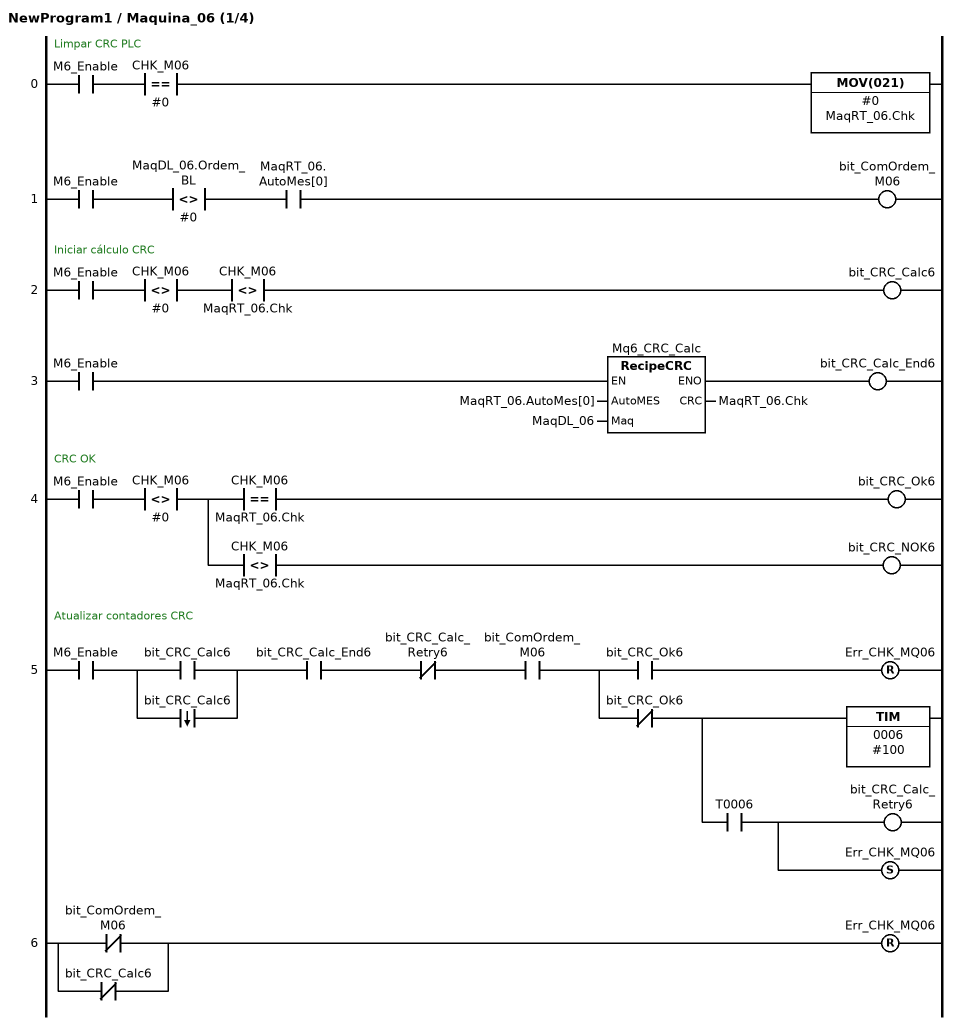
; [picture p24: NewProgram1 / Maquina_06, rungs 0-6]
; rung 0: Limpar CRC PLC
LD M6_Enable
AND=(300) CHK_M06 #0
MOV(021) #0 MaqRT_06.Chk
; rung 1
LD M6_Enable
AND<>L(306) MaqDL_06.Ordem_BL #0
AND MaqRT_06.AutoMes[0]
OUT bit_ComOrdem_M06
; rung 2: Iniciar cálculo CRC
LD M6_Enable
AND<>(305) CHK_M06 #0
AND<>(305) CHK_M06 MaqRT_06.Chk
OUT bit_CRC_Calc6
; rung 3
LD M6_Enable
CALL Mq6_CRC_Calc : RecipeCRC (AutoMES := MaqRT_06.AutoMes[0], Maq := MaqDL_06, CRC => MaqRT_06.Chk)
OUT bit_CRC_Calc_End6
; rung 4: CRC OK
LD M6_Enable
AND<>(305) CHK_M06 #0
OUT TR0
AND=(300) CHK_M06 MaqRT_06.Chk
OUT bit_CRC_Ok6
LD TR0
AND<>(305) CHK_M06 MaqRT_06.Chk
OUT bit_CRC_NOK6
; rung 5: Atualizar contadores CRC
LD M6_Enable
LD bit_CRC_Calc6
%OR bit_CRC_Calc6
ANDLD
AND bit_CRC_Calc_End6
ANDNOT bit_CRC_Calc_Retry6
AND bit_ComOrdem_M06
OUT TR0
AND bit_CRC_Ok6
RSET Err_CHK_MQ06
LD TR0
ANDNOT bit_CRC_Ok6
TIM 0006 #100
AND T0006
OUT bit_CRC_Calc_Retry6
SET Err_CHK_MQ06
; rung 6
LDNOT bit_ComOrdem_M06
ORNOT bit_CRC_Calc6
RSET Err_CHK_MQ06

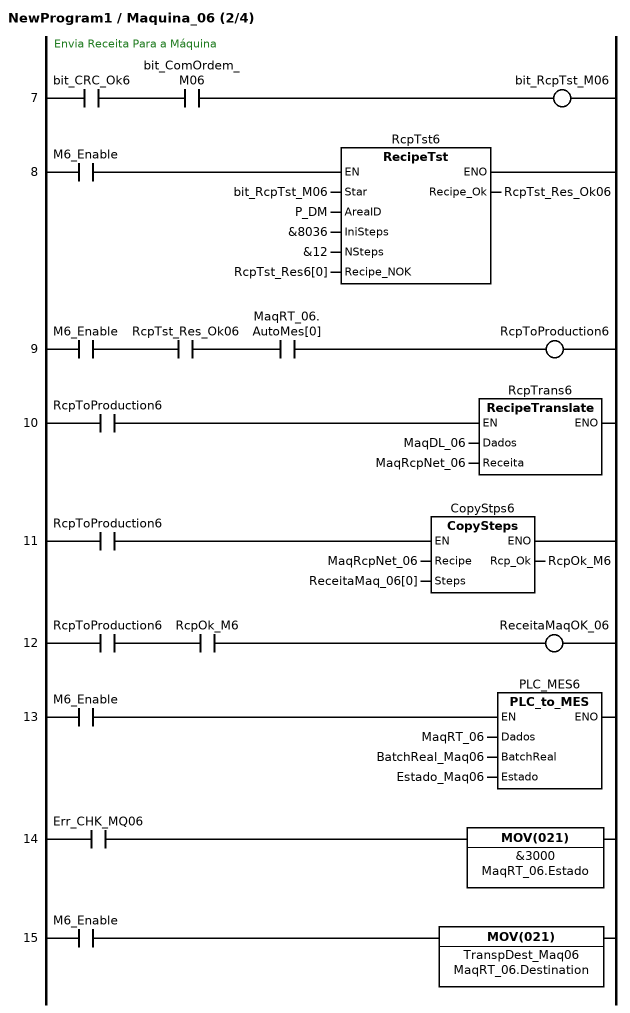
; rung 7: Envia Receita Para a Máquina
LD bit_CRC_Ok6
AND bit_ComOrdem_M06
OUT bit_RcpTst_M06
; rung 8
LD M6_Enable
CALL RcpTst6 : RecipeTst (Star := bit_RcpTst_M06, AreaID := P_DM, IniSteps := &8036, NSteps := &12, Recipe_NOK := RcpTst_Res6[0], Recipe_Ok => RcpTst_Res_Ok06)
; rung 9
LD M6_Enable
AND RcpTst_Res_Ok06
AND MaqRT_06.AutoMes[0]
OUT RcpToProduction6
; rung 10
LD RcpToProduction6
CALL RcpTrans6 : RecipeTranslate (Dados := MaqDL_06, Receita := MaqRcpNet_06)
; rung 11
LD RcpToProduction6
CALL CopyStps6 : CopySteps (Recipe := MaqRcpNet_06, Steps := ReceitaMaq_06[0], Rcp_Ok => RcpOk_M6)
; rung 12
LD RcpToProduction6
AND RcpOk_M6
OUT ReceitaMaqOK_06
; rung 13
LD M6_Enable
CALL PLC_MES6 : PLC_to_MES (Dados := MaqRT_06, BatchReal := BatchReal_Maq06, Estado := Estado_Maq06)
; rung 14
LD Err_CHK_MQ06
MOV(021) &3000 MaqRT_06.Estado
; rung 15
LD M6_Enable
MOV(021) TranspDest_Maq06 MaqRT_06.Destination

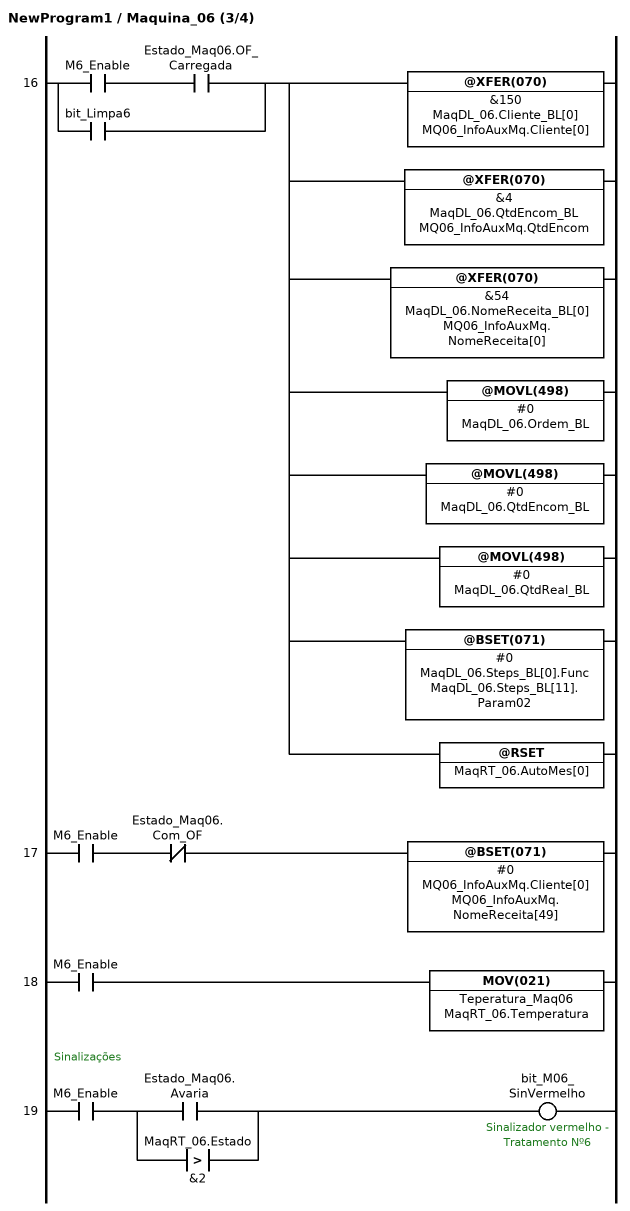
; rung 16
LD M6_Enable
AND Estado_Maq06.OF_Carregada
OR bit_Limpa6
@XFER(070) &150 MaqDL_06.Cliente_BL[0] MQ06_InfoAuxMq.Cliente[0]
@XFER(070) &4 MaqDL_06.QtdEncom_BL MQ06_InfoAuxMq.QtdEncom
@XFER(070) &54 MaqDL_06.NomeReceita_BL[0] MQ06_InfoAuxMq.NomeReceita[0]
@MOVL(498) #0 MaqDL_06.Ordem_BL
@MOVL(498) #0 MaqDL_06.QtdEncom_BL
@MOVL(498) #0 MaqDL_06.QtdReal_BL
@BSET(071) #0 MaqDL_06.Steps_BL[0].Func MaqDL_06.Steps_BL[11].Param02
@RSET MaqRT_06.AutoMes[0]
; rung 17
LD M6_Enable
ANDNOT Estado_Maq06.Com_OF
@BSET(071) #0 MQ06_InfoAuxMq.Cliente[0] MQ06_InfoAuxMq.NomeReceita[49]
; rung 18
LD M6_Enable
MOV(021) Teperatura_Maq06 MaqRT_06.Temperatura
; rung 19: Sinalizações
LD M6_Enable
LD Estado_Maq06.Avaria
OR>(320) MaqRT_06.Estado &2
ANDLD
OUT bit_M06_SinVermelho  ; Sinalizador vermelho - Tratamento Nº6

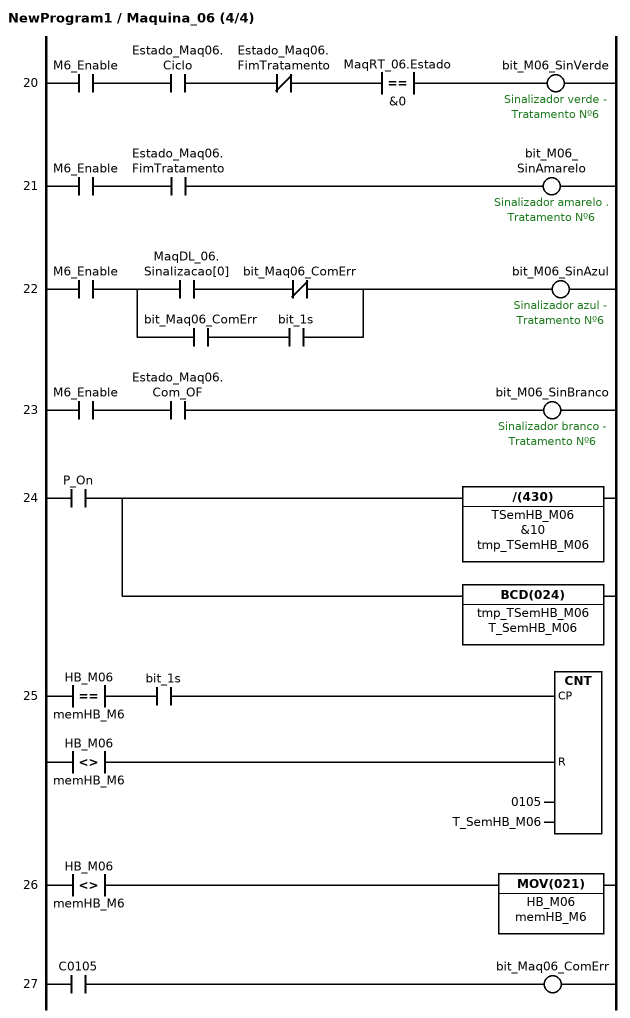
; rung 20
LD M6_Enable
AND Estado_Maq06.Ciclo
ANDNOT Estado_Maq06.FimTratamento
AND=(300) MaqRT_06.Estado &0
OUT bit_M06_SinVerde  ; Sinalizador verde - Tratamento Nº6
; rung 21
LD M6_Enable
AND Estado_Maq06.FimTratamento
OUT bit_M06_SinAmarelo  ; Sinalizador amarelo . Tratamento Nº6
; rung 22
LD M6_Enable
LD MaqDL_06.Sinalizacao[0]
ANDNOT bit_Maq06_ComErr
LD bit_Maq06_ComErr
AND bit_1s
ORLD
ANDLD
OUT bit_M06_SinAzul  ; Sinalizador azul - Tratamento Nº6
; rung 23
LD M6_Enable
AND Estado_Maq06.Com_OF
OUT bit_M06_SinBranco  ; Sinalizador branco - Tratamento Nº6
; rung 24
LD P_On
/(430) TSemHB_M06 &10 tmp_TSemHB_M06
BCD(024) tmp_TSemHB_M06 T_SemHB_M06
; rung 25
LD=(300) HB_M06 memHB_M6
AND bit_1s
LD<>(305) HB_M06 memHB_M6
CNT 0105 T_SemHB_M06
; rung 26
LD<>(305) HB_M06 memHB_M6
MOV(021) HB_M06 memHB_M6
; rung 27
LD C0105
OUT bit_Maq06_ComErr

### Section Maquina_07

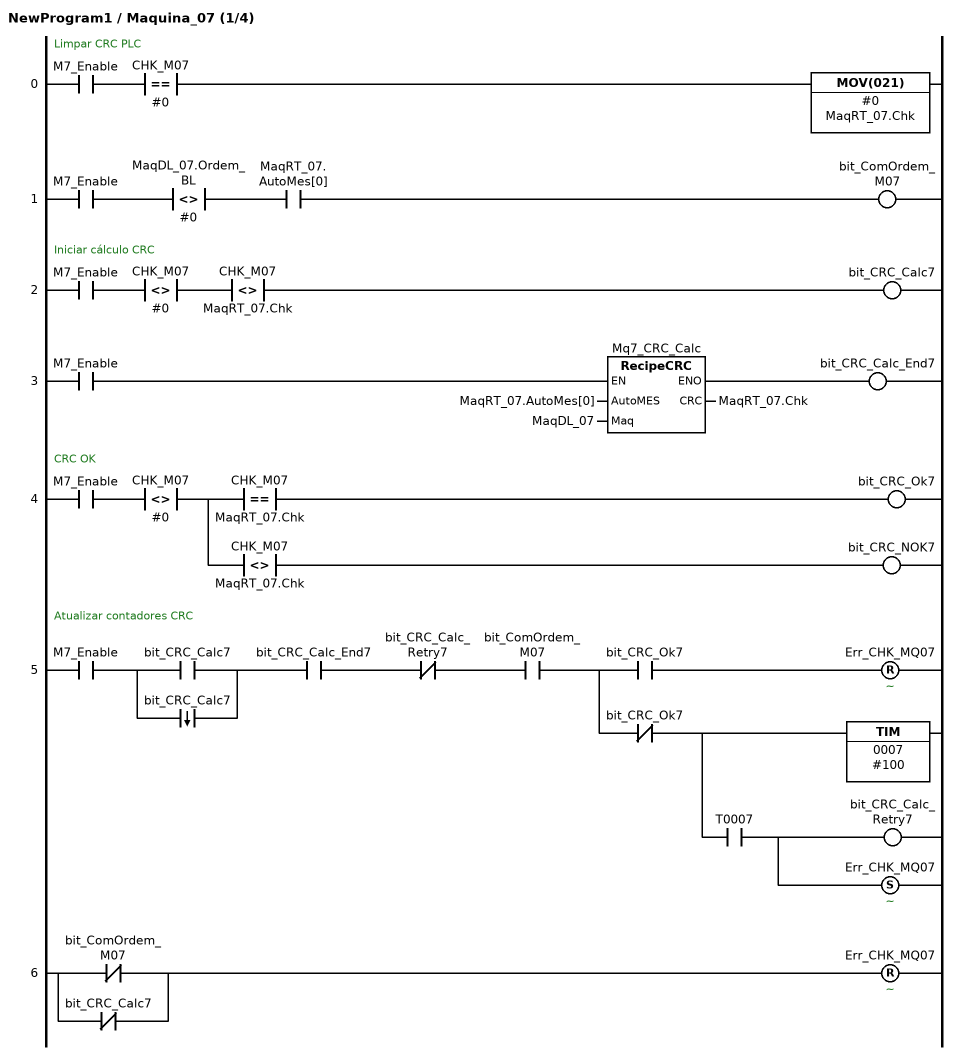
; rung 0: Limpar CRC PLC
LD M7_Enable
AND=(300) CHK_M07 #0
MOV(021) #0 MaqRT_07.Chk
; rung 1
LD M7_Enable
AND<>L(306) MaqDL_07.Ordem_BL #0
AND MaqRT_07.AutoMes[0]
OUT bit_ComOrdem_M07
; rung 2: Iniciar cálculo CRC
LD M7_Enable
AND<>(305) CHK_M07 #0
AND<>(305) CHK_M07 MaqRT_07.Chk
OUT bit_CRC_Calc7
; rung 3
LD M7_Enable
CALL Mq7_CRC_Calc : RecipeCRC (AutoMES := MaqRT_07.AutoMes[0], Maq := MaqDL_07, CRC => MaqRT_07.Chk)
OUT bit_CRC_Calc_End7
; rung 4: CRC OK
LD M7_Enable
AND<>(305) CHK_M07 #0
OUT TR0
AND=(300) CHK_M07 MaqRT_07.Chk
OUT bit_CRC_Ok7
LD TR0
AND<>(305) CHK_M07 MaqRT_07.Chk
OUT bit_CRC_NOK7
; rung 5: Atualizar contadores CRC
LD M7_Enable
LD bit_CRC_Calc7
%OR bit_CRC_Calc7
ANDLD
AND bit_CRC_Calc_End7
ANDNOT bit_CRC_Calc_Retry7
AND bit_ComOrdem_M07
OUT TR0
AND bit_CRC_Ok7
RSET Err_CHK_MQ07  ; ~
LD TR0
ANDNOT bit_CRC_Ok7
TIM 0007 #100
AND T0007
OUT bit_CRC_Calc_Retry7
SET Err_CHK_MQ07  ; ~
; rung 6
LDNOT bit_ComOrdem_M07
ORNOT bit_CRC_Calc7
RSET Err_CHK_MQ07  ; ~

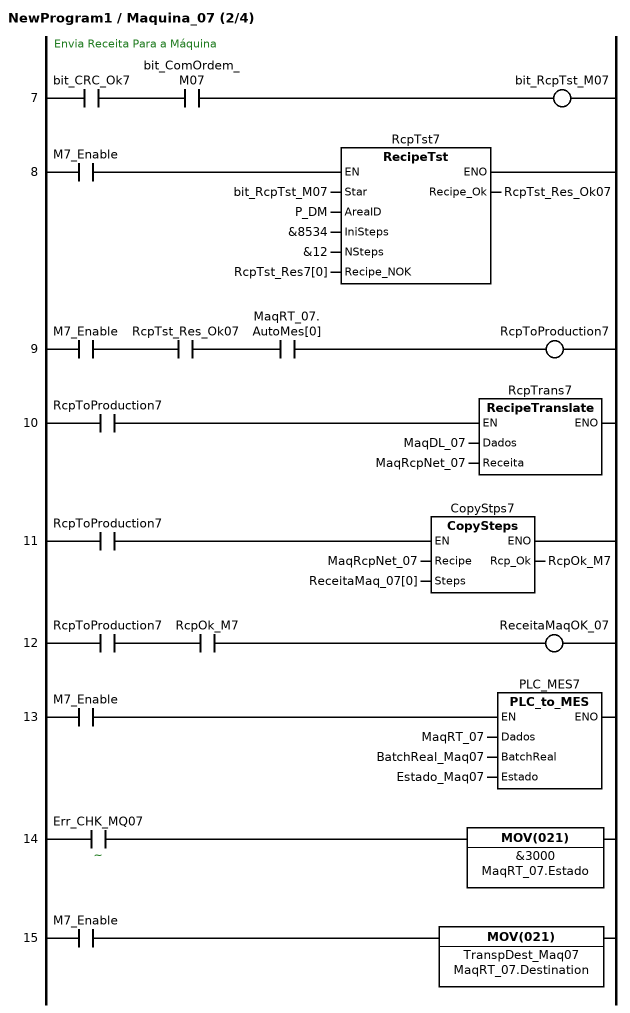
; rung 7: Envia Receita Para a Máquina
LD bit_CRC_Ok7
AND bit_ComOrdem_M07
OUT bit_RcpTst_M07
; rung 8
LD M7_Enable
CALL RcpTst7 : RecipeTst (Star := bit_RcpTst_M07, AreaID := P_DM, IniSteps := &8534, NSteps := &12, Recipe_NOK := RcpTst_Res7[0], Recipe_Ok => RcpTst_Res_Ok07)
; rung 9
LD M7_Enable
AND RcpTst_Res_Ok07
AND MaqRT_07.AutoMes[0]
OUT RcpToProduction7
; rung 10
LD RcpToProduction7
CALL RcpTrans7 : RecipeTranslate (Dados := MaqDL_07, Receita := MaqRcpNet_07)
; rung 11
LD RcpToProduction7
CALL CopyStps7 : CopySteps (Recipe := MaqRcpNet_07, Steps := ReceitaMaq_07[0], Rcp_Ok => RcpOk_M7)
; rung 12
LD RcpToProduction7
AND RcpOk_M7
OUT ReceitaMaqOK_07
; rung 13
LD M7_Enable
CALL PLC_MES7 : PLC_to_MES (Dados := MaqRT_07, BatchReal := BatchReal_Maq07, Estado := Estado_Maq07)
; rung 14
LD Err_CHK_MQ07  ; ~
MOV(021) &3000 MaqRT_07.Estado
; rung 15
LD M7_Enable
MOV(021) TranspDest_Maq07 MaqRT_07.Destination

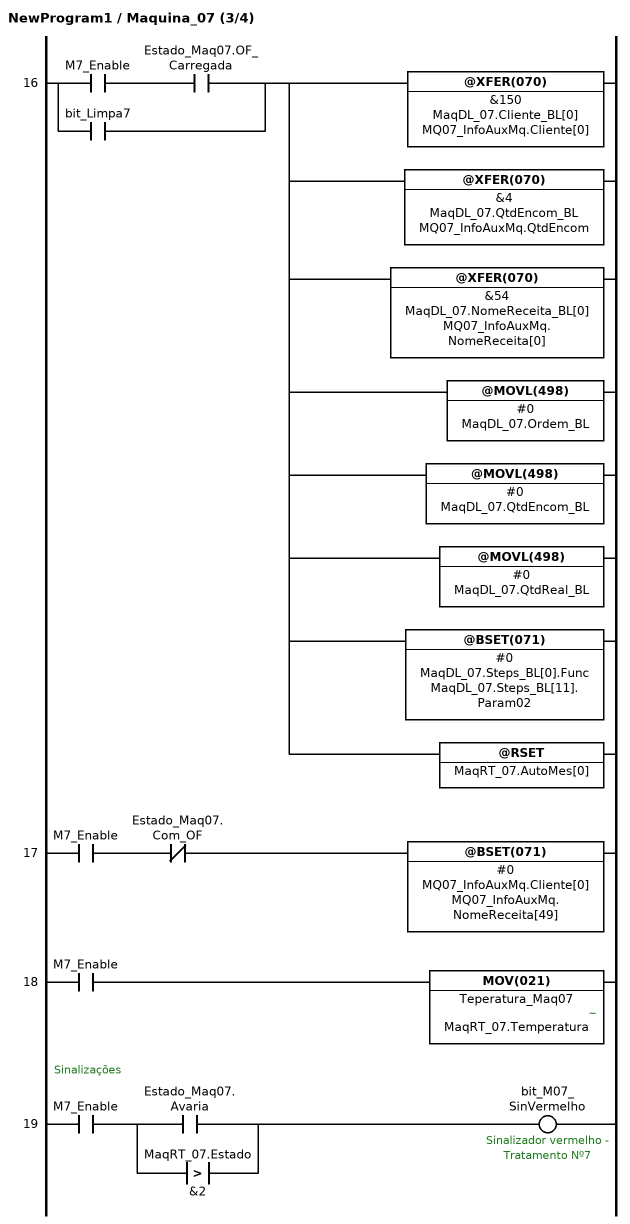
; rung 16
LD M7_Enable
AND Estado_Maq07.OF_Carregada
OR bit_Limpa7
@XFER(070) &150 MaqDL_07.Cliente_BL[0] MQ07_InfoAuxMq.Cliente[0]
@XFER(070) &4 MaqDL_07.QtdEncom_BL MQ07_InfoAuxMq.QtdEncom
@XFER(070) &54 MaqDL_07.NomeReceita_BL[0] MQ07_InfoAuxMq.NomeReceita[0]
@MOVL(498) #0 MaqDL_07.Ordem_BL
@MOVL(498) #0 MaqDL_07.QtdEncom_BL
@MOVL(498) #0 MaqDL_07.QtdReal_BL
@BSET(071) #0 MaqDL_07.Steps_BL[0].Func MaqDL_07.Steps_BL[11].Param02
@RSET MaqRT_07.AutoMes[0]
; rung 17
LD M7_Enable
ANDNOT Estado_Maq07.Com_OF
@BSET(071) #0 MQ07_InfoAuxMq.Cliente[0] MQ07_InfoAuxMq.NomeReceita[49]
; rung 18
LD M7_Enable
MOV(021) Teperatura_Maq07 MaqRT_07.Temperatura  ; ~
; rung 19: Sinalizações
LD M7_Enable
LD Estado_Maq07.Avaria
OR>(320) MaqRT_07.Estado &2
ANDLD
OUT bit_M07_SinVermelho  ; Sinalizador vermelho - Tratamento Nº7

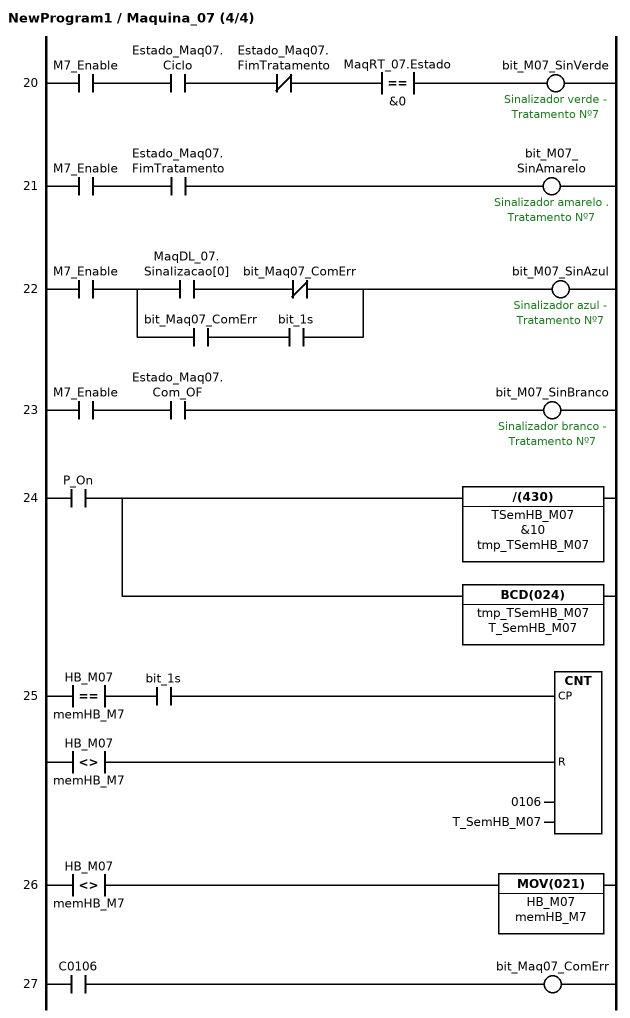
; rung 20
LD M7_Enable
AND Estado_Maq07.Ciclo
ANDNOT Estado_Maq07.FimTratamento
AND=(300) MaqRT_07.Estado &0
OUT bit_M07_SinVerde  ; Sinalizador verde - Tratamento Nº7
; rung 21
LD M7_Enable
AND Estado_Maq07.FimTratamento
OUT bit_M07_SinAmarelo  ; Sinalizador amarelo . Tratamento Nº7
; rung 22
LD M7_Enable
LD MaqDL_07.Sinalizacao[0]
ANDNOT bit_Maq07_ComErr
LD bit_Maq07_ComErr
AND bit_1s
ORLD
ANDLD
OUT bit_M07_SinAzul  ; Sinalizador azul - Tratamento Nº7
; rung 23
LD M7_Enable
AND Estado_Maq07.Com_OF
OUT bit_M07_SinBranco  ; Sinalizador branco - Tratamento Nº7
; rung 24
LD P_On
/(430) TSemHB_M07 &10 tmp_TSemHB_M07
BCD(024) tmp_TSemHB_M07 T_SemHB_M07
; rung 25
LD=(300) HB_M07 memHB_M7
AND bit_1s
LD<>(305) HB_M07 memHB_M7
CNT 0106 T_SemHB_M07
; rung 26
LD<>(305) HB_M07 memHB_M7
MOV(021) HB_M07 memHB_M7
; rung 27
LD C0106
OUT bit_Maq07_ComErr

### Section Maquina_08

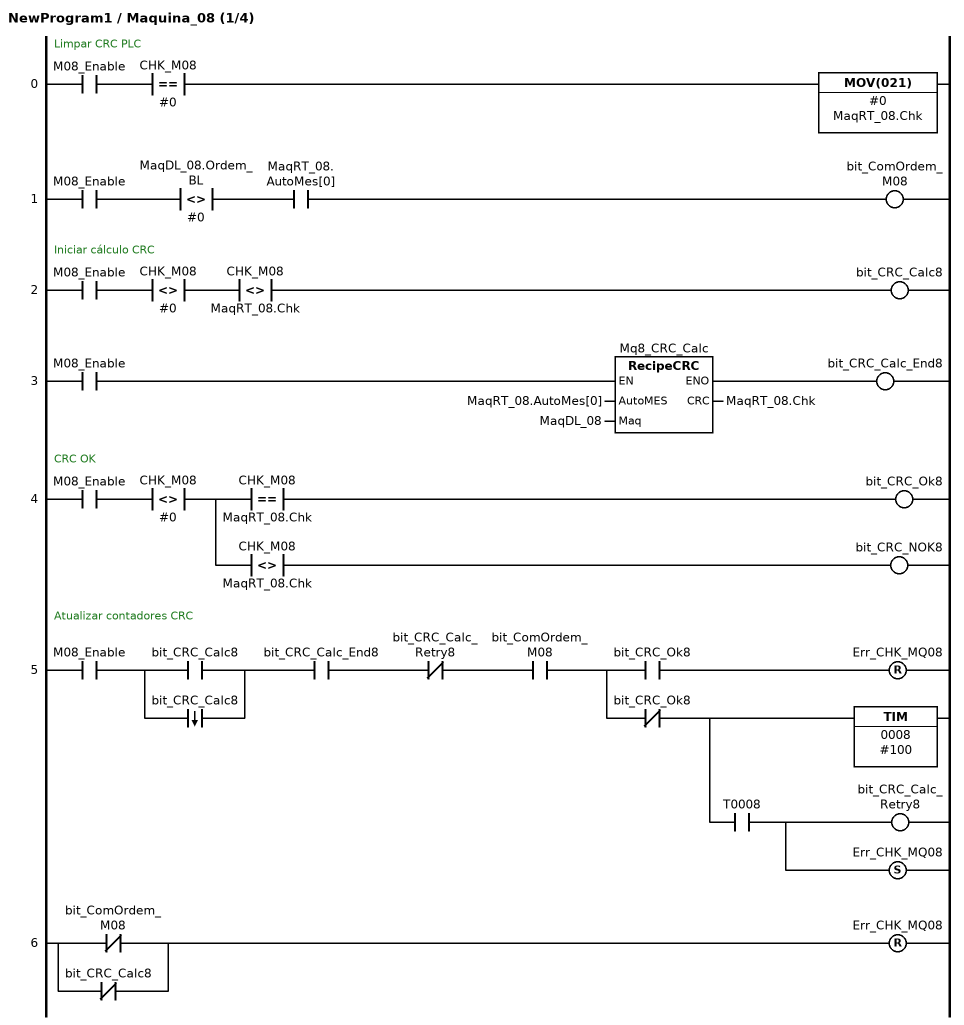
; rung 0: Limpar CRC PLC
LD M08_Enable
AND=(300) CHK_M08 #0
MOV(021) #0 MaqRT_08.Chk
; rung 1
LD M08_Enable
AND<>L(306) MaqDL_08.Ordem_BL #0
AND MaqRT_08.AutoMes[0]
OUT bit_ComOrdem_M08
; rung 2: Iniciar cálculo CRC
LD M08_Enable
AND<>(305) CHK_M08 #0
AND<>(305) CHK_M08 MaqRT_08.Chk
OUT bit_CRC_Calc8
; rung 3
LD M08_Enable
CALL Mq8_CRC_Calc : RecipeCRC (AutoMES := MaqRT_08.AutoMes[0], Maq := MaqDL_08, CRC => MaqRT_08.Chk)
OUT bit_CRC_Calc_End8
; rung 4: CRC OK
LD M08_Enable
AND<>(305) CHK_M08 #0
OUT TR0
AND=(300) CHK_M08 MaqRT_08.Chk
OUT bit_CRC_Ok8
LD TR0
AND<>(305) CHK_M08 MaqRT_08.Chk
OUT bit_CRC_NOK8
; rung 5: Atualizar contadores CRC
LD M08_Enable
LD bit_CRC_Calc8
%OR bit_CRC_Calc8
ANDLD
AND bit_CRC_Calc_End8
ANDNOT bit_CRC_Calc_Retry8
AND bit_ComOrdem_M08
OUT TR0
AND bit_CRC_Ok8
RSET Err_CHK_MQ08
LD TR0
ANDNOT bit_CRC_Ok8
TIM 0008 #100
AND T0008
OUT bit_CRC_Calc_Retry8
SET Err_CHK_MQ08
; rung 6
LDNOT bit_ComOrdem_M08
ORNOT bit_CRC_Calc8
RSET Err_CHK_MQ08

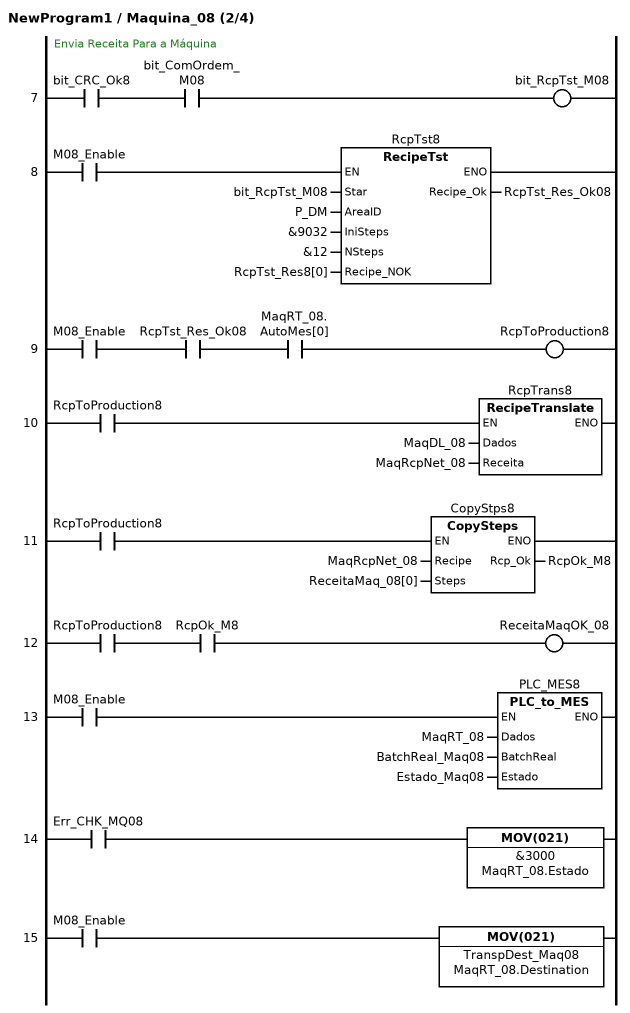
; rung 7: Envia Receita Para a Máquina
LD bit_CRC_Ok8
AND bit_ComOrdem_M08
OUT bit_RcpTst_M08
; rung 8
LD M08_Enable
CALL RcpTst8 : RecipeTst (Star := bit_RcpTst_M08, AreaID := P_DM, IniSteps := &9032, NSteps := &12, Recipe_NOK := RcpTst_Res8[0], Recipe_Ok => RcpTst_Res_Ok08)
; rung 9
LD M08_Enable
AND RcpTst_Res_Ok08
AND MaqRT_08.AutoMes[0]
OUT RcpToProduction8
; rung 10
LD RcpToProduction8
CALL RcpTrans8 : RecipeTranslate (Dados := MaqDL_08, Receita := MaqRcpNet_08)
; rung 11
LD RcpToProduction8
CALL CopyStps8 : CopySteps (Recipe := MaqRcpNet_08, Steps := ReceitaMaq_08[0], Rcp_Ok => RcpOk_M8)
; rung 12
LD RcpToProduction8
AND RcpOk_M8
OUT ReceitaMaqOK_08
; rung 13
LD M08_Enable
CALL PLC_MES8 : PLC_to_MES (Dados := MaqRT_08, BatchReal := BatchReal_Maq08, Estado := Estado_Maq08)
; rung 14
LD Err_CHK_MQ08
MOV(021) &3000 MaqRT_08.Estado
; rung 15
LD M08_Enable
MOV(021) TranspDest_Maq08 MaqRT_08.Destination

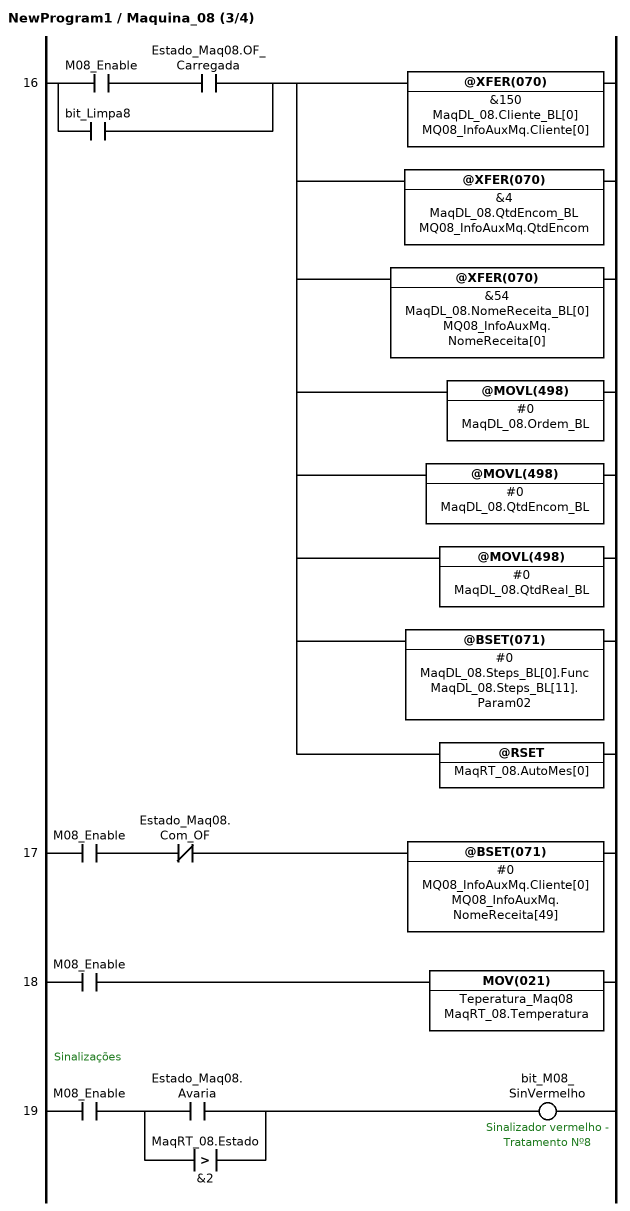
; rung 16
LD M08_Enable
AND Estado_Maq08.OF_Carregada
OR bit_Limpa8
@XFER(070) &150 MaqDL_08.Cliente_BL[0] MQ08_InfoAuxMq.Cliente[0]
@XFER(070) &4 MaqDL_08.QtdEncom_BL MQ08_InfoAuxMq.QtdEncom
@XFER(070) &54 MaqDL_08.NomeReceita_BL[0] MQ08_InfoAuxMq.NomeReceita[0]
@MOVL(498) #0 MaqDL_08.Ordem_BL
@MOVL(498) #0 MaqDL_08.QtdEncom_BL
@MOVL(498) #0 MaqDL_08.QtdReal_BL
@BSET(071) #0 MaqDL_08.Steps_BL[0].Func MaqDL_08.Steps_BL[11].Param02
@RSET MaqRT_08.AutoMes[0]
; rung 17
LD M08_Enable
ANDNOT Estado_Maq08.Com_OF
@BSET(071) #0 MQ08_InfoAuxMq.Cliente[0] MQ08_InfoAuxMq.NomeReceita[49]
; rung 18
LD M08_Enable
MOV(021) Teperatura_Maq08 MaqRT_08.Temperatura
; rung 19: Sinalizações
LD M08_Enable
LD Estado_Maq08.Avaria
OR>(320) MaqRT_08.Estado &2
ANDLD
OUT bit_M08_SinVermelho  ; Sinalizador vermelho - Tratamento Nº8

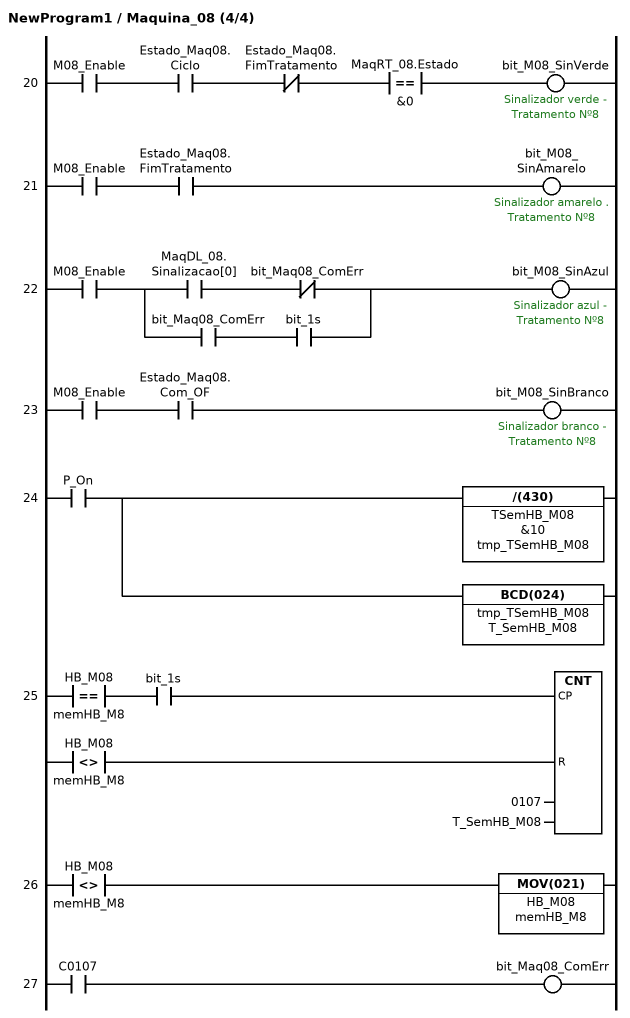
; rung 20
LD M08_Enable
AND Estado_Maq08.Ciclo
ANDNOT Estado_Maq08.FimTratamento
AND=(300) MaqRT_08.Estado &0
OUT bit_M08_SinVerde  ; Sinalizador verde - Tratamento Nº8
; rung 21
LD M08_Enable
AND Estado_Maq08.FimTratamento
OUT bit_M08_SinAmarelo  ; Sinalizador amarelo . Tratamento Nº8
; rung 22
LD M08_Enable
LD MaqDL_08.Sinalizacao[0]
ANDNOT bit_Maq08_ComErr
LD bit_Maq08_ComErr
AND bit_1s
ORLD
ANDLD
OUT bit_M08_SinAzul  ; Sinalizador azul - Tratamento Nº8
; rung 23
LD M08_Enable
AND Estado_Maq08.Com_OF
OUT bit_M08_SinBranco  ; Sinalizador branco - Tratamento Nº8
; rung 24
LD P_On
/(430) TSemHB_M08 &10 tmp_TSemHB_M08
BCD(024) tmp_TSemHB_M08 T_SemHB_M08
; rung 25
LD=(300) HB_M08 memHB_M8
AND bit_1s
LD<>(305) HB_M08 memHB_M8
CNT 0107 T_SemHB_M08
; rung 26
LD<>(305) HB_M08 memHB_M8
MOV(021) HB_M08 memHB_M8
; rung 27
LD C0107
OUT bit_Maq08_ComErr

### Section Maquina_09

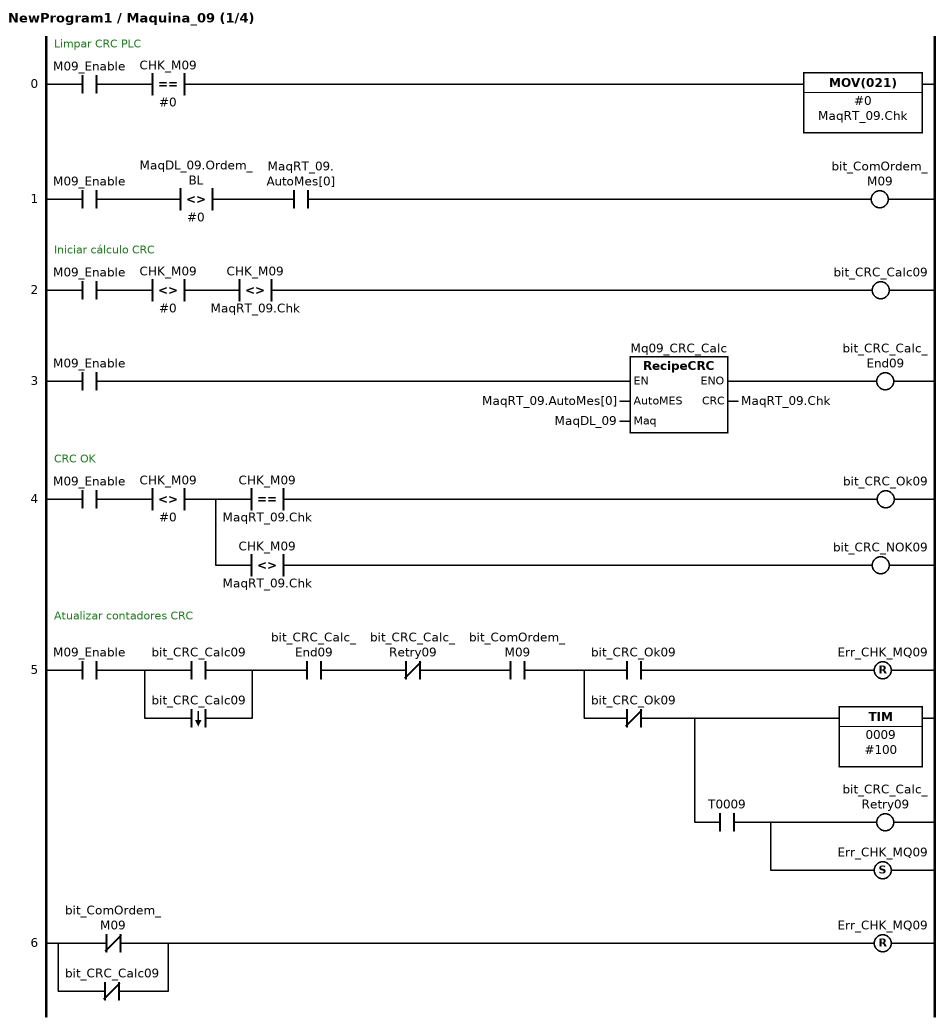
; rung 0: Limpar CRC PLC
LD M09_Enable
AND=(300) CHK_M09 #0
MOV(021) #0 MaqRT_09.Chk
; rung 1
LD M09_Enable
AND<>L(306) MaqDL_09.Ordem_BL #0
AND MaqRT_09.AutoMes[0]
OUT bit_ComOrdem_M09
; rung 2: Iniciar cálculo CRC
LD M09_Enable
AND<>(305) CHK_M09 #0
AND<>(305) CHK_M09 MaqRT_09.Chk
OUT bit_CRC_Calc09
; rung 3
LD M09_Enable
CALL Mq09_CRC_Calc : RecipeCRC (AutoMES := MaqRT_09.AutoMes[0], Maq := MaqDL_09, CRC => MaqRT_09.Chk)
OUT bit_CRC_Calc_End09
; rung 4: CRC OK
LD M09_Enable
AND<>(305) CHK_M09 #0
OUT TR0
AND=(300) CHK_M09 MaqRT_09.Chk
OUT bit_CRC_Ok09
LD TR0
AND<>(305) CHK_M09 MaqRT_09.Chk
OUT bit_CRC_NOK09
; rung 5: Atualizar contadores CRC
LD M09_Enable
LD bit_CRC_Calc09
%OR bit_CRC_Calc09
ANDLD
AND bit_CRC_Calc_End09
ANDNOT bit_CRC_Calc_Retry09
AND bit_ComOrdem_M09
OUT TR0
AND bit_CRC_Ok09
RSET Err_CHK_MQ09
LD TR0
ANDNOT bit_CRC_Ok09
TIM 0009 #100
AND T0009
OUT bit_CRC_Calc_Retry09
SET Err_CHK_MQ09
; rung 6
LDNOT bit_ComOrdem_M09
ORNOT bit_CRC_Calc09
RSET Err_CHK_MQ09

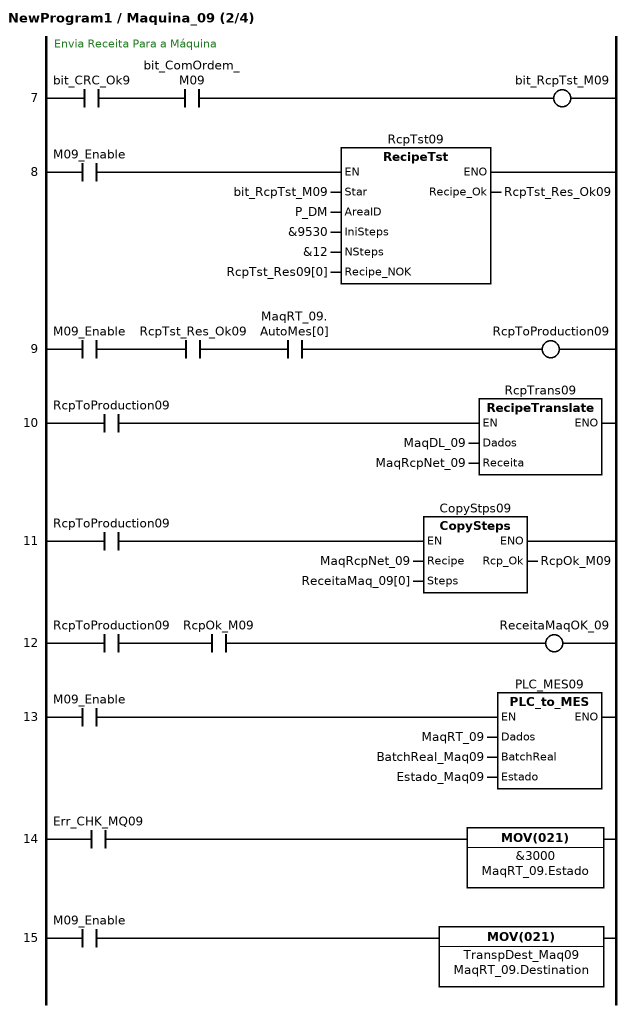
; rung 7: Envia Receita Para a Máquina
LD bit_CRC_Ok9
AND bit_ComOrdem_M09
OUT bit_RcpTst_M09
; rung 8
LD M09_Enable
CALL RcpTst09 : RecipeTst (Star := bit_RcpTst_M09, AreaID := P_DM, IniSteps := &9530, NSteps := &12, Recipe_NOK := RcpTst_Res09[0], Recipe_Ok => RcpTst_Res_Ok09)
; rung 9
LD M09_Enable
AND RcpTst_Res_Ok09
AND MaqRT_09.AutoMes[0]
OUT RcpToProduction09
; rung 10
LD RcpToProduction09
CALL RcpTrans09 : RecipeTranslate (Dados := MaqDL_09, Receita := MaqRcpNet_09)
; rung 11
LD RcpToProduction09
CALL CopyStps09 : CopySteps (Recipe := MaqRcpNet_09, Steps := ReceitaMaq_09[0], Rcp_Ok => RcpOk_M09)
; rung 12
LD RcpToProduction09
AND RcpOk_M09
OUT ReceitaMaqOK_09
; rung 13
LD M09_Enable
CALL PLC_MES09 : PLC_to_MES (Dados := MaqRT_09, BatchReal := BatchReal_Maq09, Estado := Estado_Maq09)
; rung 14
LD Err_CHK_MQ09
MOV(021) &3000 MaqRT_09.Estado
; rung 15
LD M09_Enable
MOV(021) TranspDest_Maq09 MaqRT_09.Destination

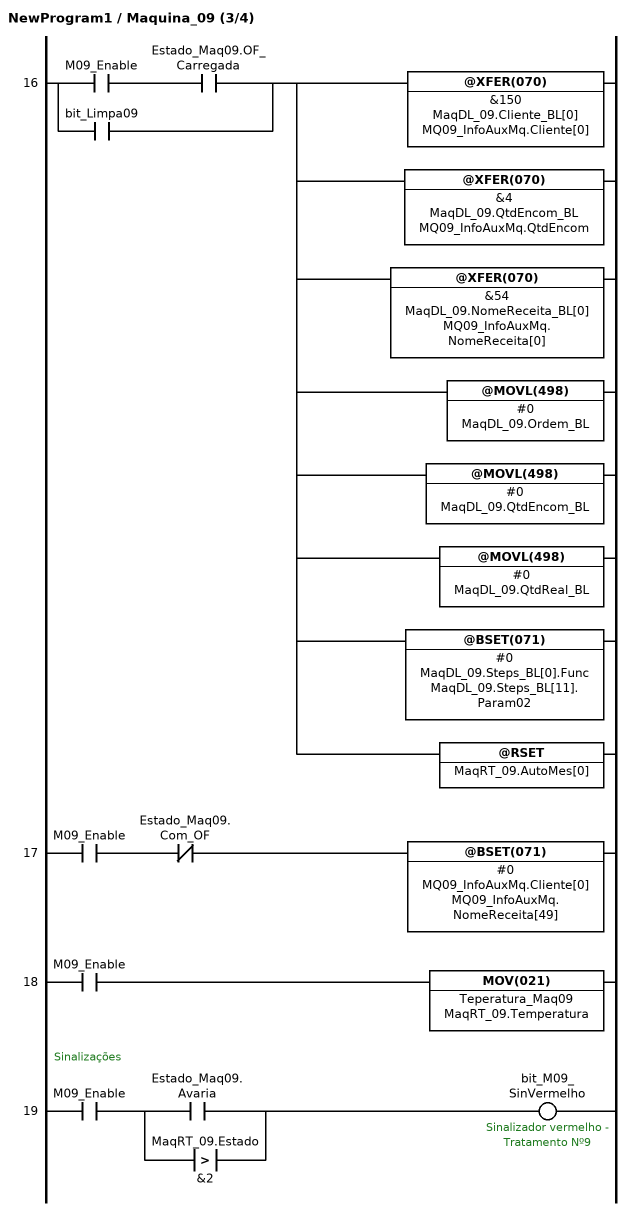
; rung 16
LD M09_Enable
AND Estado_Maq09.OF_Carregada
OR bit_Limpa09
@XFER(070) &150 MaqDL_09.Cliente_BL[0] MQ09_InfoAuxMq.Cliente[0]
@XFER(070) &4 MaqDL_09.QtdEncom_BL MQ09_InfoAuxMq.QtdEncom
@XFER(070) &54 MaqDL_09.NomeReceita_BL[0] MQ09_InfoAuxMq.NomeReceita[0]
@MOVL(498) #0 MaqDL_09.Ordem_BL
@MOVL(498) #0 MaqDL_09.QtdEncom_BL
@MOVL(498) #0 MaqDL_09.QtdReal_BL
@BSET(071) #0 MaqDL_09.Steps_BL[0].Func MaqDL_09.Steps_BL[11].Param02
@RSET MaqRT_09.AutoMes[0]
; rung 17
LD M09_Enable
ANDNOT Estado_Maq09.Com_OF
@BSET(071) #0 MQ09_InfoAuxMq.Cliente[0] MQ09_InfoAuxMq.NomeReceita[49]
; rung 18
LD M09_Enable
MOV(021) Teperatura_Maq09 MaqRT_09.Temperatura
; rung 19: Sinalizações
LD M09_Enable
LD Estado_Maq09.Avaria
OR>(320) MaqRT_09.Estado &2
ANDLD
OUT bit_M09_SinVermelho  ; Sinalizador vermelho - Tratamento Nº9

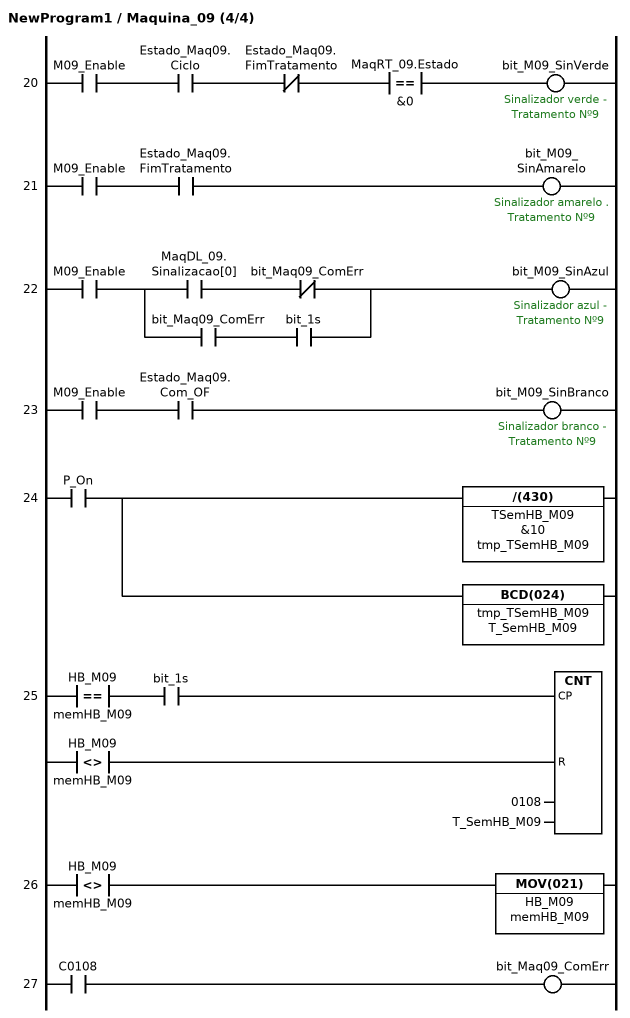
; rung 20
LD M09_Enable
AND Estado_Maq09.Ciclo
ANDNOT Estado_Maq09.FimTratamento
AND=(300) MaqRT_09.Estado &0
OUT bit_M09_SinVerde  ; Sinalizador verde - Tratamento Nº9
; rung 21
LD M09_Enable
AND Estado_Maq09.FimTratamento
OUT bit_M09_SinAmarelo  ; Sinalizador amarelo . Tratamento Nº9
; rung 22
LD M09_Enable
LD MaqDL_09.Sinalizacao[0]
ANDNOT bit_Maq09_ComErr
LD bit_Maq09_ComErr
AND bit_1s
ORLD
ANDLD
OUT bit_M09_SinAzul  ; Sinalizador azul - Tratamento Nº9
; rung 23
LD M09_Enable
AND Estado_Maq09.Com_OF
OUT bit_M09_SinBranco  ; Sinalizador branco - Tratamento Nº9
; rung 24
LD P_On
/(430) TSemHB_M09 &10 tmp_TSemHB_M09
BCD(024) tmp_TSemHB_M09 T_SemHB_M09
; rung 25
LD=(300) HB_M09 memHB_M09
AND bit_1s
LD<>(305) HB_M09 memHB_M09
CNT 0108 T_SemHB_M09
; rung 26
LD<>(305) HB_M09 memHB_M09
MOV(021) HB_M09 memHB_M09
; rung 27
LD C0108
OUT bit_Maq09_ComErr

### Section Maquina_10

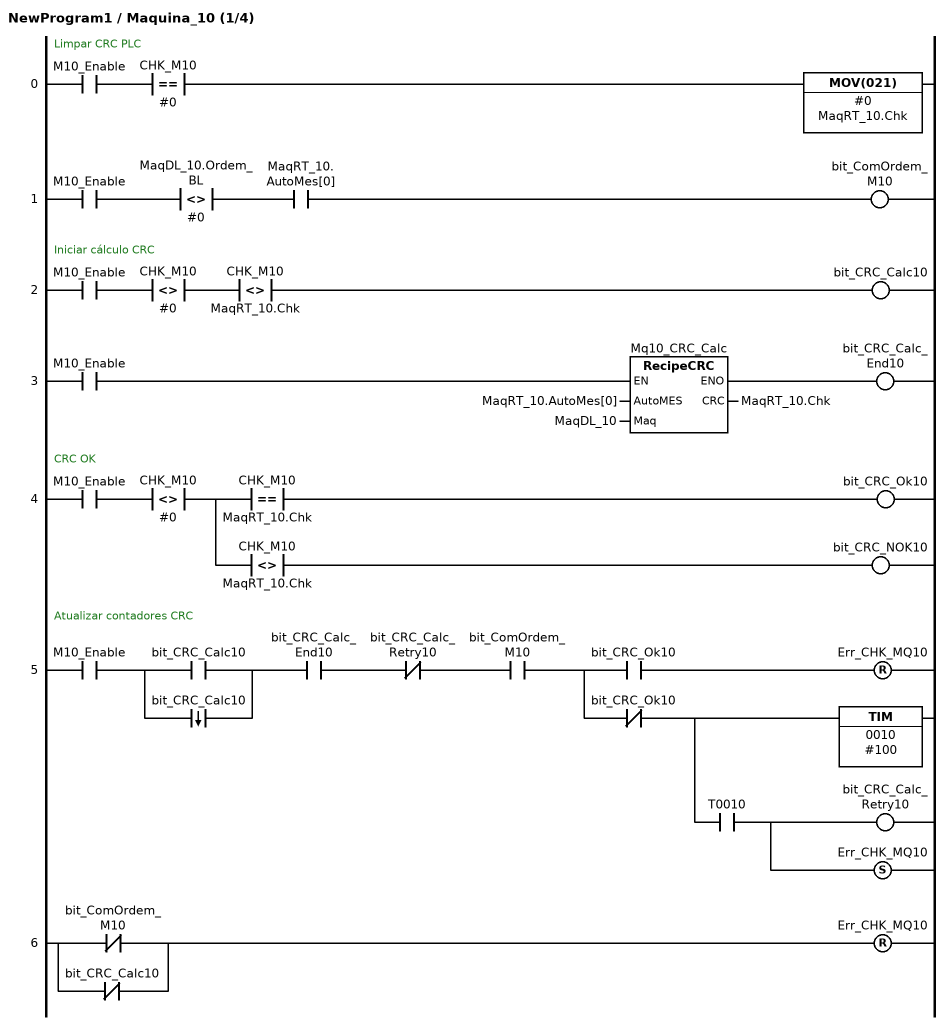
; rung 0: Limpar CRC PLC
LD M10_Enable
AND=(300) CHK_M10 #0
MOV(021) #0 MaqRT_10.Chk
; rung 1
LD M10_Enable
AND<>L(306) MaqDL_10.Ordem_BL #0
AND MaqRT_10.AutoMes[0]
OUT bit_ComOrdem_M10
; rung 2: Iniciar cálculo CRC
LD M10_Enable
AND<>(305) CHK_M10 #0
AND<>(305) CHK_M10 MaqRT_10.Chk
OUT bit_CRC_Calc10
; rung 3
LD M10_Enable
CALL Mq10_CRC_Calc : RecipeCRC (AutoMES := MaqRT_10.AutoMes[0], Maq := MaqDL_10, CRC => MaqRT_10.Chk)
OUT bit_CRC_Calc_End10
; rung 4: CRC OK
LD M10_Enable
AND<>(305) CHK_M10 #0
OUT TR0
AND=(300) CHK_M10 MaqRT_10.Chk
OUT bit_CRC_Ok10
LD TR0
AND<>(305) CHK_M10 MaqRT_10.Chk
OUT bit_CRC_NOK10
; rung 5: Atualizar contadores CRC
LD M10_Enable
LD bit_CRC_Calc10
%OR bit_CRC_Calc10
ANDLD
AND bit_CRC_Calc_End10
ANDNOT bit_CRC_Calc_Retry10
AND bit_ComOrdem_M10
OUT TR0
AND bit_CRC_Ok10
RSET Err_CHK_MQ10
LD TR0
ANDNOT bit_CRC_Ok10
TIM 0010 #100
AND T0010
OUT bit_CRC_Calc_Retry10
SET Err_CHK_MQ10
; rung 6
LDNOT bit_ComOrdem_M10
ORNOT bit_CRC_Calc10
RSET Err_CHK_MQ10

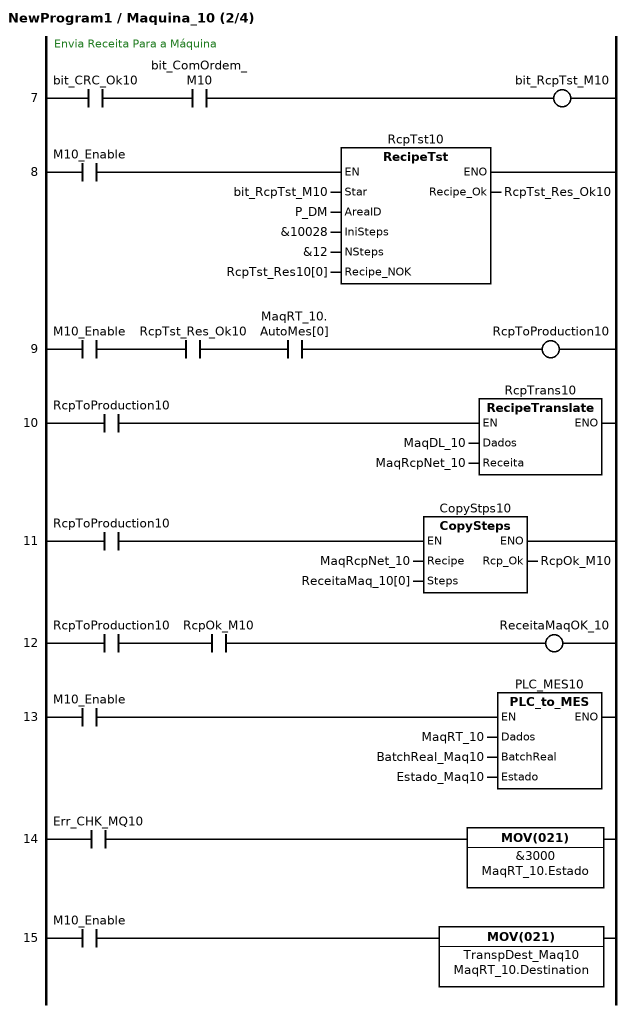
; rung 7: Envia Receita Para a Máquina
LD bit_CRC_Ok10
AND bit_ComOrdem_M10
OUT bit_RcpTst_M10
; rung 8
LD M10_Enable
CALL RcpTst10 : RecipeTst (Star := bit_RcpTst_M10, AreaID := P_DM, IniSteps := &10028, NSteps := &12, Recipe_NOK := RcpTst_Res10[0], Recipe_Ok => RcpTst_Res_Ok10)
; rung 9
LD M10_Enable
AND RcpTst_Res_Ok10
AND MaqRT_10.AutoMes[0]
OUT RcpToProduction10
; rung 10
LD RcpToProduction10
CALL RcpTrans10 : RecipeTranslate (Dados := MaqDL_10, Receita := MaqRcpNet_10)
; rung 11
LD RcpToProduction10
CALL CopyStps10 : CopySteps (Recipe := MaqRcpNet_10, Steps := ReceitaMaq_10[0], Rcp_Ok => RcpOk_M10)
; rung 12
LD RcpToProduction10
AND RcpOk_M10
OUT ReceitaMaqOK_10
; rung 13
LD M10_Enable
CALL PLC_MES10 : PLC_to_MES (Dados := MaqRT_10, BatchReal := BatchReal_Maq10, Estado := Estado_Maq10)
; rung 14
LD Err_CHK_MQ10
MOV(021) &3000 MaqRT_10.Estado
; rung 15
LD M10_Enable
MOV(021) TranspDest_Maq10 MaqRT_10.Destination

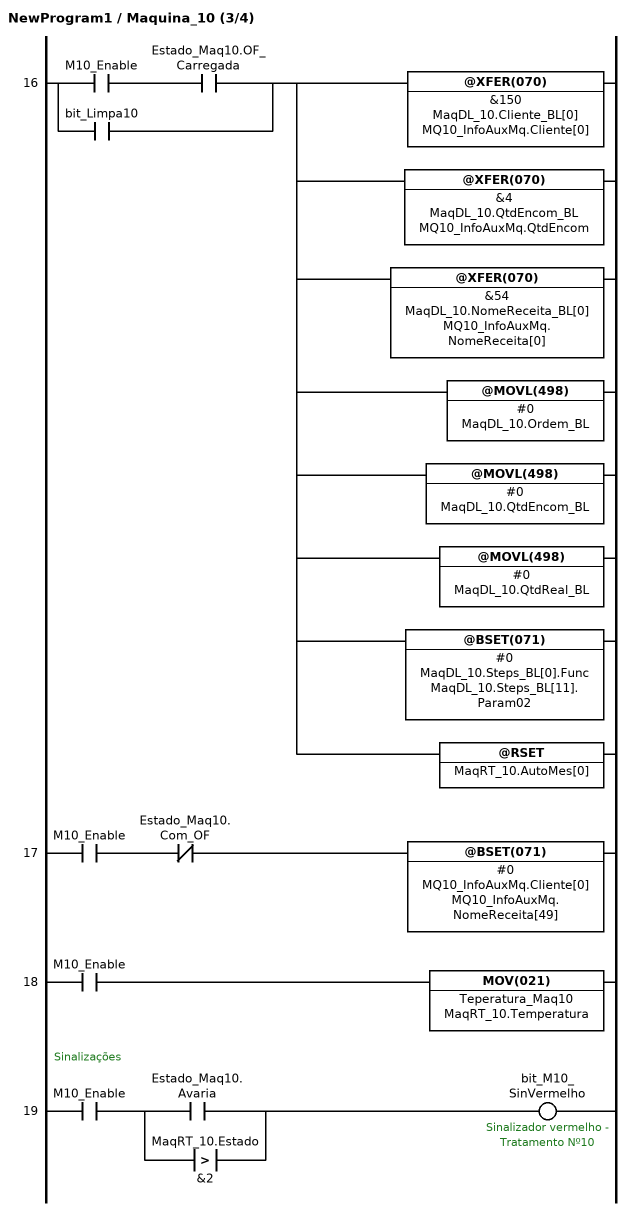
; rung 16
LD M10_Enable
AND Estado_Maq10.OF_Carregada
OR bit_Limpa10
@XFER(070) &150 MaqDL_10.Cliente_BL[0] MQ10_InfoAuxMq.Cliente[0]
@XFER(070) &4 MaqDL_10.QtdEncom_BL MQ10_InfoAuxMq.QtdEncom
@XFER(070) &54 MaqDL_10.NomeReceita_BL[0] MQ10_InfoAuxMq.NomeReceita[0]
@MOVL(498) #0 MaqDL_10.Ordem_BL
@MOVL(498) #0 MaqDL_10.QtdEncom_BL
@MOVL(498) #0 MaqDL_10.QtdReal_BL
@BSET(071) #0 MaqDL_10.Steps_BL[0].Func MaqDL_10.Steps_BL[11].Param02
@RSET MaqRT_10.AutoMes[0]
; rung 17
LD M10_Enable
ANDNOT Estado_Maq10.Com_OF
@BSET(071) #0 MQ10_InfoAuxMq.Cliente[0] MQ10_InfoAuxMq.NomeReceita[49]
; rung 18
LD M10_Enable
MOV(021) Teperatura_Maq10 MaqRT_10.Temperatura
; rung 19: Sinalizações
LD M10_Enable
LD Estado_Maq10.Avaria
OR>(320) MaqRT_10.Estado &2
ANDLD
OUT bit_M10_SinVermelho  ; Sinalizador vermelho - Tratamento Nº10

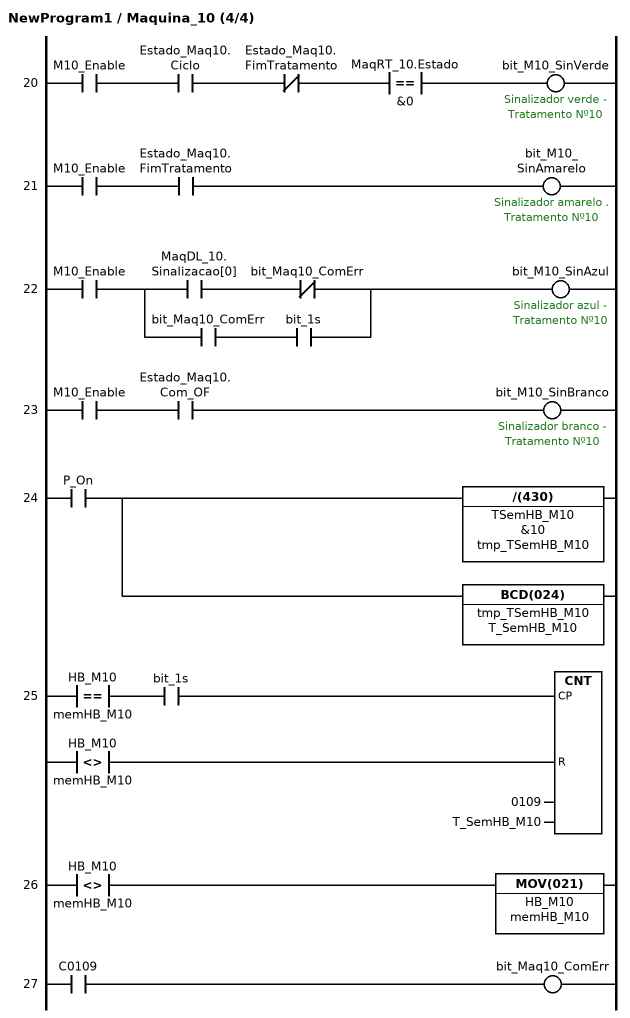
; rung 20
LD M10_Enable
AND Estado_Maq10.Ciclo
ANDNOT Estado_Maq10.FimTratamento
AND=(300) MaqRT_10.Estado &0
OUT bit_M10_SinVerde  ; Sinalizador verde - Tratamento Nº10
; rung 21
LD M10_Enable
AND Estado_Maq10.FimTratamento
OUT bit_M10_SinAmarelo  ; Sinalizador amarelo . Tratamento Nº10
; rung 22
LD M10_Enable
LD MaqDL_10.Sinalizacao[0]
ANDNOT bit_Maq10_ComErr
LD bit_Maq10_ComErr
AND bit_1s
ORLD
ANDLD
OUT bit_M10_SinAzul  ; Sinalizador azul - Tratamento Nº10
; rung 23
LD M10_Enable
AND Estado_Maq10.Com_OF
OUT bit_M10_SinBranco  ; Sinalizador branco - Tratamento Nº10
; rung 24
LD P_On
/(430) TSemHB_M10 &10 tmp_TSemHB_M10
BCD(024) tmp_TSemHB_M10 T_SemHB_M10
; rung 25
LD=(300) HB_M10 memHB_M10
AND bit_1s
LD<>(305) HB_M10 memHB_M10
CNT 0109 T_SemHB_M10
; rung 26
LD<>(305) HB_M10 memHB_M10
MOV(021) HB_M10 memHB_M10
; rung 27
LD C0109
OUT bit_Maq10_ComErr

### Section Maquina_11

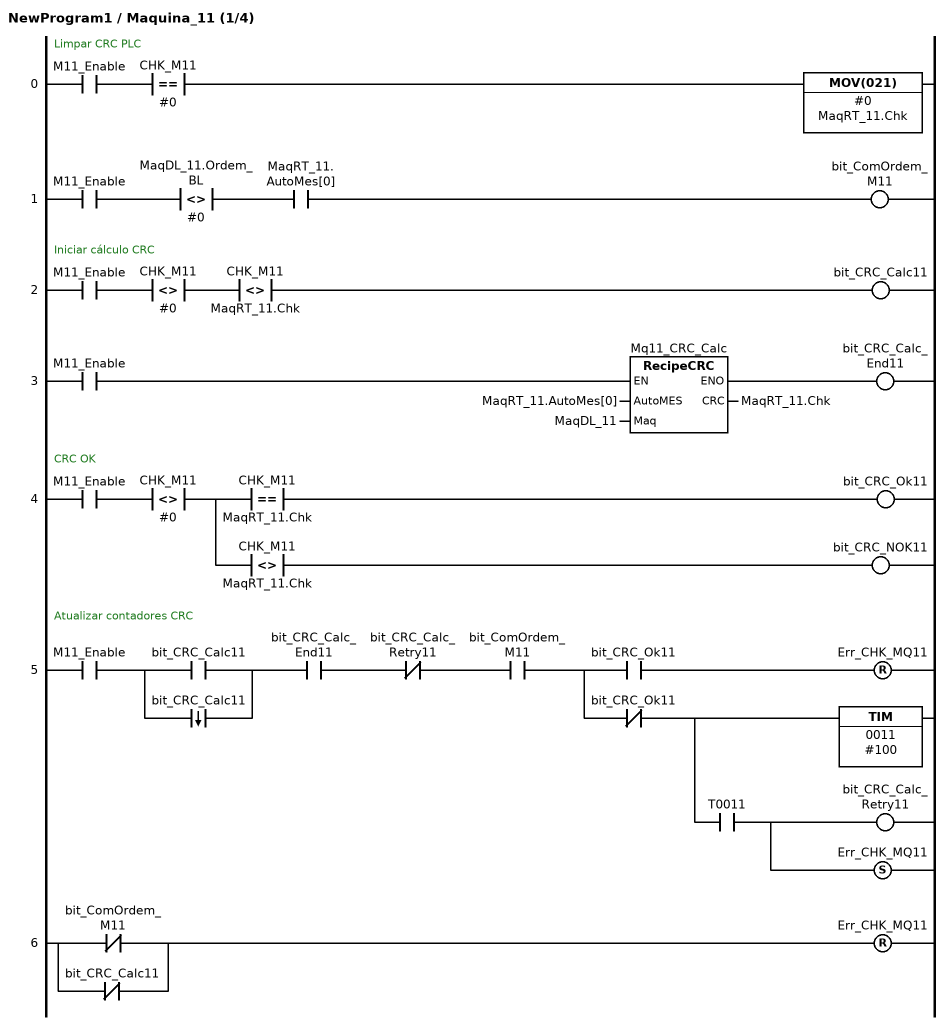
; rung 0: Limpar CRC PLC
LD M11_Enable
AND=(300) CHK_M11 #0
MOV(021) #0 MaqRT_11.Chk
; rung 1
LD M11_Enable
AND<>L(306) MaqDL_11.Ordem_BL #0
AND MaqRT_11.AutoMes[0]
OUT bit_ComOrdem_M11
; rung 2: Iniciar cálculo CRC
LD M11_Enable
AND<>(305) CHK_M11 #0
AND<>(305) CHK_M11 MaqRT_11.Chk
OUT bit_CRC_Calc11
; rung 3
LD M11_Enable
CALL Mq11_CRC_Calc : RecipeCRC (AutoMES := MaqRT_11.AutoMes[0], Maq := MaqDL_11, CRC => MaqRT_11.Chk)
OUT bit_CRC_Calc_End11
; rung 4: CRC OK
LD M11_Enable
AND<>(305) CHK_M11 #0
OUT TR0
AND=(300) CHK_M11 MaqRT_11.Chk
OUT bit_CRC_Ok11
LD TR0
AND<>(305) CHK_M11 MaqRT_11.Chk
OUT bit_CRC_NOK11
; rung 5: Atualizar contadores CRC
LD M11_Enable
LD bit_CRC_Calc11
%OR bit_CRC_Calc11
ANDLD
AND bit_CRC_Calc_End11
ANDNOT bit_CRC_Calc_Retry11
AND bit_ComOrdem_M11
OUT TR0
AND bit_CRC_Ok11
RSET Err_CHK_MQ11
LD TR0
ANDNOT bit_CRC_Ok11
TIM 0011 #100
AND T0011
OUT bit_CRC_Calc_Retry11
SET Err_CHK_MQ11
; rung 6
LDNOT bit_ComOrdem_M11
ORNOT bit_CRC_Calc11
RSET Err_CHK_MQ11

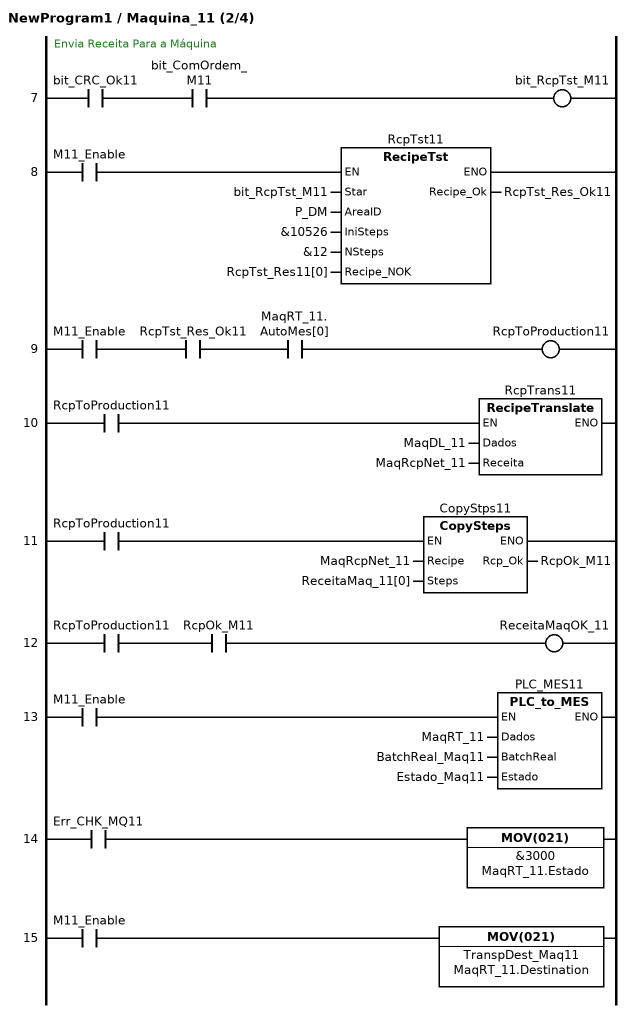
; rung 7: Envia Receita Para a Máquina
LD bit_CRC_Ok11
AND bit_ComOrdem_M11
OUT bit_RcpTst_M11
; rung 8
LD M11_Enable
CALL RcpTst11 : RecipeTst (Star := bit_RcpTst_M11, AreaID := P_DM, IniSteps := &10526, NSteps := &12, Recipe_NOK := RcpTst_Res11[0], Recipe_Ok => RcpTst_Res_Ok11)
; rung 9
LD M11_Enable
AND RcpTst_Res_Ok11
AND MaqRT_11.AutoMes[0]
OUT RcpToProduction11
; rung 10
LD RcpToProduction11
CALL RcpTrans11 : RecipeTranslate (Dados := MaqDL_11, Receita := MaqRcpNet_11)
; rung 11
LD RcpToProduction11
CALL CopyStps11 : CopySteps (Recipe := MaqRcpNet_11, Steps := ReceitaMaq_11[0], Rcp_Ok => RcpOk_M11)
; rung 12
LD RcpToProduction11
AND RcpOk_M11
OUT ReceitaMaqOK_11
; rung 13
LD M11_Enable
CALL PLC_MES11 : PLC_to_MES (Dados := MaqRT_11, BatchReal := BatchReal_Maq11, Estado := Estado_Maq11)
; rung 14
LD Err_CHK_MQ11
MOV(021) &3000 MaqRT_11.Estado
; rung 15
LD M11_Enable
MOV(021) TranspDest_Maq11 MaqRT_11.Destination

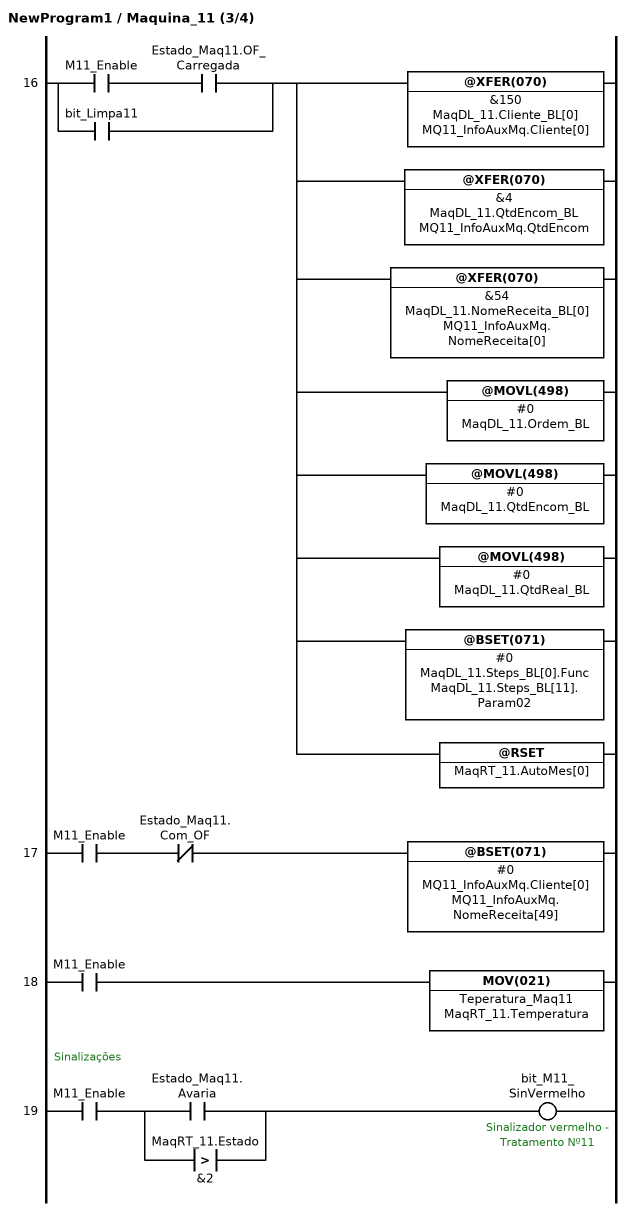
; rung 16
LD M11_Enable
AND Estado_Maq11.OF_Carregada
OR bit_Limpa11
@XFER(070) &150 MaqDL_11.Cliente_BL[0] MQ11_InfoAuxMq.Cliente[0]
@XFER(070) &4 MaqDL_11.QtdEncom_BL MQ11_InfoAuxMq.QtdEncom
@XFER(070) &54 MaqDL_11.NomeReceita_BL[0] MQ11_InfoAuxMq.NomeReceita[0]
@MOVL(498) #0 MaqDL_11.Ordem_BL
@MOVL(498) #0 MaqDL_11.QtdEncom_BL
@MOVL(498) #0 MaqDL_11.QtdReal_BL
@BSET(071) #0 MaqDL_11.Steps_BL[0].Func MaqDL_11.Steps_BL[11].Param02
@RSET MaqRT_11.AutoMes[0]
; rung 17
LD M11_Enable
ANDNOT Estado_Maq11.Com_OF
@BSET(071) #0 MQ11_InfoAuxMq.Cliente[0] MQ11_InfoAuxMq.NomeReceita[49]
; rung 18
LD M11_Enable
MOV(021) Teperatura_Maq11 MaqRT_11.Temperatura
; rung 19: Sinalizações
LD M11_Enable
LD Estado_Maq11.Avaria
OR>(320) MaqRT_11.Estado &2
ANDLD
OUT bit_M11_SinVermelho  ; Sinalizador vermelho - Tratamento Nº11

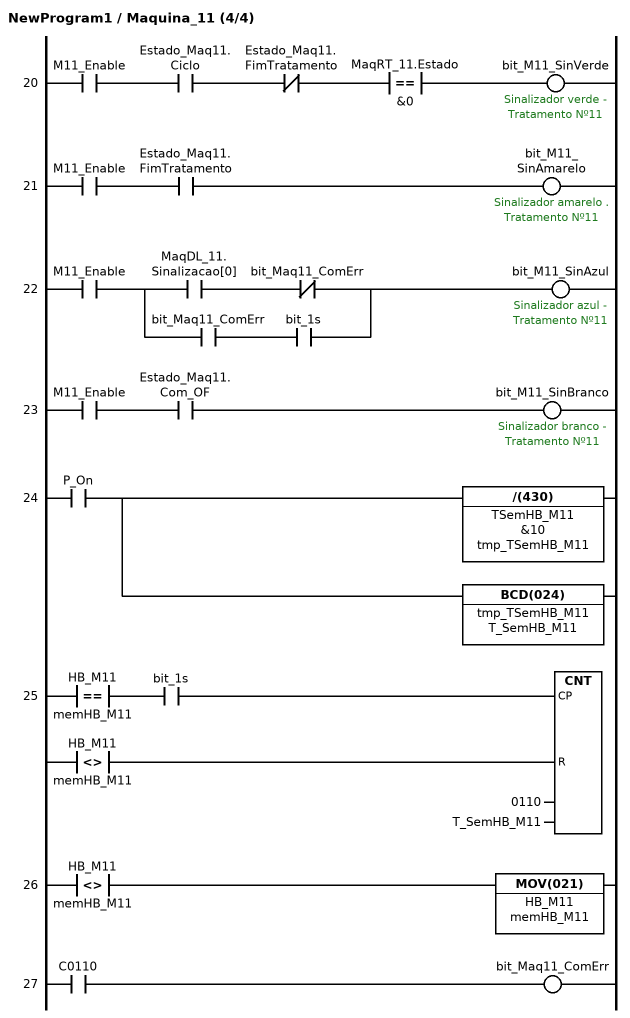
; rung 20
LD M11_Enable
AND Estado_Maq11.Ciclo
ANDNOT Estado_Maq11.FimTratamento
AND=(300) MaqRT_11.Estado &0
OUT bit_M11_SinVerde  ; Sinalizador verde - Tratamento Nº11
; rung 21
LD M11_Enable
AND Estado_Maq11.FimTratamento
OUT bit_M11_SinAmarelo  ; Sinalizador amarelo . Tratamento Nº11
; rung 22
LD M11_Enable
LD MaqDL_11.Sinalizacao[0]
ANDNOT bit_Maq11_ComErr
LD bit_Maq11_ComErr
AND bit_1s
ORLD
ANDLD
OUT bit_M11_SinAzul  ; Sinalizador azul - Tratamento Nº11
; rung 23
LD M11_Enable
AND Estado_Maq11.Com_OF
OUT bit_M11_SinBranco  ; Sinalizador branco - Tratamento Nº11
; rung 24
LD P_On
/(430) TSemHB_M11 &10 tmp_TSemHB_M11
BCD(024) tmp_TSemHB_M11 T_SemHB_M11
; rung 25
LD=(300) HB_M11 memHB_M11
AND bit_1s
LD<>(305) HB_M11 memHB_M11
CNT 0110 T_SemHB_M11
; rung 26
LD<>(305) HB_M11 memHB_M11
MOV(021) HB_M11 memHB_M11
; rung 27
LD C0110
OUT bit_Maq11_ComErr

### Section Sinalizacao

